// TIA Portal V17 export
// export: Created 2024-09-03T21:54:54.8850339Z, ExportSetting WithDefaults, DisplayName Totally Integrated Automation Portal, DisplayVersion V17 Update 7, DisplayName TIA Portal Openness, DisplayVersion V17 Update 7, DisplayName TIA Portal Version Control Interface, DisplayVersion V17, DisplayName SINAMICS Startdrive Advanced, DisplayVersion V17 SP2, DisplayName SINAMICS Startdrive G110M, G120, G120C, G120D, G120P, G115D, DisplayVersion V17 SP2, DisplayName SINAMICS Startdrive G130, G150, S120, S150, SINAMICS MV, S210, DisplayVersion V17 SP2, DisplayName STEP 7 Professional, DisplayVersion V17 Update 7, DisplayName STEP 7 Safety, DisplayVersion V17 Update 6, DisplayName WinCC Advanced / Unified PC, DisplayVersion V17 Update 7
DATA_BLOCK "DB_ProductionProgramList"   // DB6100
{ S7_Optimized_Access := 'FALSE' }
VERSION : 0.1
// stored: AutoNumber false, DBAccessibleFromOPCUA true, DBAccessibleFromWebserver true, IsOnlyStoredInLoadMemory false, IsWriteProtectedInAS false
   VAR RETAIN
      Program { S7_SetPoint := 'True'} : Array[1.."NumberOfProductionPrograms"] of "UDT_ProductionProgram";
   END_VAR
BEGIN
   Program[1]."Name" := 'LH-6 way';
   Program[2]."Name" := 'RH-6 way';
   Program[3]."Name" := 'LH-4 way';
   Program[4]."Name" := 'RH-4 way';
   Program[5]."Name" := 'startup';
   Program[6]."Name" := 'startup RH';
   Program[7..8]."Name" := '';
   Program[1].CupformingParametersLeft.DigiforceProgram := 1;
   Program[2].CupformingParametersLeft.DigiforceProgram := 2;
   Program[3].CupformingParametersLeft.DigiforceProgram := 1;
   Program[4].CupformingParametersLeft.DigiforceProgram := 2;
   Program[5..6].CupformingParametersLeft.DigiforceProgram := 1;
   Program[7..8].CupformingParametersLeft.DigiforceProgram := 0;
   Program[1..2].CupformingParametersLeft.FinalSpeed := 30.0;
   Program[3].CupformingParametersLeft.FinalSpeed := 20.0;
   Program[4].CupformingParametersLeft.FinalSpeed := 30.0;
   Program[5].CupformingParametersLeft.FinalSpeed := 25.0;
   Program[6].CupformingParametersLeft.FinalSpeed := 20.0;
   Program[7..8].CupformingParametersLeft.FinalSpeed := 0.0;
   Program[1..2].CupformingParametersLeft.ApproachSpeed := 95.0;
   Program[3].CupformingParametersLeft.ApproachSpeed := 100.0;
   Program[4].CupformingParametersLeft.ApproachSpeed := 95.0;
   Program[5].CupformingParametersLeft.ApproachSpeed := 25.0;
   Program[6].CupformingParametersLeft.ApproachSpeed := 100.0;
   Program[7..8].CupformingParametersLeft.ApproachSpeed := 0.0;
   Program[1..4].CupformingParametersLeft.FinalForce := 90.0;
   Program[5].CupformingParametersLeft.FinalForce := 10.0;
   Program[6].CupformingParametersLeft.FinalForce := 90.0;
   Program[7..8].CupformingParametersLeft.FinalForce := 0.0;
   Program[1..4].CupformingParametersLeft.ApproachForce := 20.0;
   Program[5].CupformingParametersLeft.ApproachForce := 10.0;
   Program[6].CupformingParametersLeft.ApproachForce := 20.0;
   Program[7..8].CupformingParametersLeft.ApproachForce := 0.0;
   Program[1..4].CupformingParametersLeft.EndWayImmediate := 7.5;
   Program[5].CupformingParametersLeft.EndWayImmediate := 2.55;
   Program[6].CupformingParametersLeft.EndWayImmediate := 9.9;
   Program[7..8].CupformingParametersLeft.EndWayImmediate := 0.0;
   Program[1..4].CupformingParametersLeft.EndWayWithTimeout := 8.6;
   Program[5].CupformingParametersLeft.EndWayWithTimeout := 3.0;
   Program[6].CupformingParametersLeft.EndWayWithTimeout := 9.9;
   Program[7..8].CupformingParametersLeft.EndWayWithTimeout := 0.0;
   Program[1..4].CupformingParametersLeft.SwitchingWay := 50.0;
   Program[5].CupformingParametersLeft.SwitchingWay := 20.0;
   Program[6].CupformingParametersLeft.SwitchingWay := 50.0;
   Program[7..8].CupformingParametersLeft.SwitchingWay := 0.0;
   Program[1..5].CupformingParametersLeft.EndWayTimeout := T#300MS;
   Program[6].CupformingParametersLeft.EndWayTimeout := T#200MS;
   Program[7..8].CupformingParametersLeft.EndWayTimeout := T#0MS;
   Program[1].CupformingParametersRight.DigiforceProgram := 1;
   Program[2].CupformingParametersRight.DigiforceProgram := 2;
   Program[3].CupformingParametersRight.DigiforceProgram := 1;
   Program[4].CupformingParametersRight.DigiforceProgram := 2;
   Program[5..6].CupformingParametersRight.DigiforceProgram := 1;
   Program[7..8].CupformingParametersRight.DigiforceProgram := 0;
   Program[1..4].CupformingParametersRight.FinalSpeed := 30.0;
   Program[5].CupformingParametersRight.FinalSpeed := 25.0;
   Program[6].CupformingParametersRight.FinalSpeed := 20.0;
   Program[7..8].CupformingParametersRight.FinalSpeed := 0.0;
   Program[1..2].CupformingParametersRight.ApproachSpeed := 100.0;
   Program[3].CupformingParametersRight.ApproachSpeed := 95.0;
   Program[4].CupformingParametersRight.ApproachSpeed := 100.0;
   Program[5].CupformingParametersRight.ApproachSpeed := 25.0;
   Program[6].CupformingParametersRight.ApproachSpeed := 100.0;
   Program[7..8].CupformingParametersRight.ApproachSpeed := 0.0;
   Program[1..6].CupformingParametersRight.FinalForce := 60.0;
   Program[7..8].CupformingParametersRight.FinalForce := 0.0;
   Program[1..6].CupformingParametersRight.ApproachForce := 10.0;
   Program[7..8].CupformingParametersRight.ApproachForce := 0.0;
   Program[1..4].CupformingParametersRight.EndWayImmediate := 7.8;
   Program[5].CupformingParametersRight.EndWayImmediate := 2.7;
   Program[6].CupformingParametersRight.EndWayImmediate := 9.9;
   Program[7..8].CupformingParametersRight.EndWayImmediate := 0.0;
   Program[1..2].CupformingParametersRight.EndWayWithTimeout := 8.4;
   Program[3].CupformingParametersRight.EndWayWithTimeout := 8.6;
   Program[4].CupformingParametersRight.EndWayWithTimeout := 8.4;
   Program[5].CupformingParametersRight.EndWayWithTimeout := 3.0;
   Program[6].CupformingParametersRight.EndWayWithTimeout := 9.9;
   Program[7..8].CupformingParametersRight.EndWayWithTimeout := 0.0;
   Program[1..4].CupformingParametersRight.SwitchingWay := 50.0;
   Program[5].CupformingParametersRight.SwitchingWay := 20.0;
   Program[6].CupformingParametersRight.SwitchingWay := 50.0;
   Program[7..8].CupformingParametersRight.SwitchingWay := 0.0;
   Program[1..4].CupformingParametersRight.EndWayTimeout := T#1S;
   Program[5].CupformingParametersRight.EndWayTimeout := T#300MS;
   Program[6].CupformingParametersRight.EndWayTimeout := T#200MS;
   Program[7..8].CupformingParametersRight.EndWayTimeout := T#0MS;
   Program[1].St1Insertion[1..6] := TRUE;
   Program[1].St1Insertion[7..20] := FALSE;
   Program[2].St1Insertion[1..6] := TRUE;
   Program[2].St1Insertion[7..20] := FALSE;
   Program[3].St1Insertion[1..2] := TRUE;
   Program[3].St1Insertion[3] := FALSE;
   Program[3].St1Insertion[4..6] := TRUE;
   Program[3].St1Insertion[7..20] := FALSE;
   Program[4].St1Insertion[1..5] := TRUE;
   Program[4].St1Insertion[6..20] := FALSE;
   Program[5].St1Insertion[1] := TRUE;
   Program[5].St1Insertion[2] := FALSE;
   Program[5].St1Insertion[3..5] := TRUE;
   Program[5].St1Insertion[6] := FALSE;
   Program[5].St1Insertion[7] := TRUE;
   Program[5].St1Insertion[8] := FALSE;
   Program[5].St1Insertion[9..10] := TRUE;
   Program[5].St1Insertion[11] := FALSE;
   Program[5].St1Insertion[12..17] := TRUE;
   Program[5].St1Insertion[18] := FALSE;
   Program[5].St1Insertion[19] := TRUE;
   Program[5].St1Insertion[20] := FALSE;
   Program[6].St1Insertion[1..4] := TRUE;
   Program[6].St1Insertion[5..20] := FALSE;
   Program[7].St1Insertion[1..20] := FALSE;
   Program[8].St1Insertion[1..20] := FALSE;
   Program[1].St1InsertionUsed[1..6] := TRUE;
   Program[1].St1InsertionUsed[7..20] := FALSE;
   Program[2].St1InsertionUsed[1..6] := TRUE;
   Program[2].St1InsertionUsed[7..20] := FALSE;
   Program[3].St1InsertionUsed[1..2] := TRUE;
   Program[3].St1InsertionUsed[3] := FALSE;
   Program[3].St1InsertionUsed[4..6] := TRUE;
   Program[3].St1InsertionUsed[7..20] := FALSE;
   Program[4].St1InsertionUsed[1..5] := TRUE;
   Program[4].St1InsertionUsed[6..20] := FALSE;
   Program[5].St1InsertionUsed[1..7] := TRUE;
   Program[5].St1InsertionUsed[8] := FALSE;
   Program[5].St1InsertionUsed[9..19] := TRUE;
   Program[5].St1InsertionUsed[20] := FALSE;
   Program[6].St1InsertionUsed[1..4] := TRUE;
   Program[6].St1InsertionUsed[5..20] := FALSE;
   Program[7].St1InsertionUsed[1..20] := FALSE;
   Program[8].St1InsertionUsed[1..20] := FALSE;
   Program[1].FaureciaNumber := '2824317X';
   Program[2].FaureciaNumber := '2841135X';
   Program[3].FaureciaNumber := '2824317X';
   Program[4].FaureciaNumber := '2841135X';
   Program[5].FaureciaNumber := '2567208X';
   Program[6].FaureciaNumber := 'xxxx';
   Program[7..8].FaureciaNumber := '';
   Program[1..6].FaureciaNumberStartChar := 9;
   Program[7..8].FaureciaNumberStartChar := 0;
   Program[1..6].FaureciaNumberLength := 8;
   Program[7..8].FaureciaNumberLength := 0;
   Program[1].MechanicalType := 0;
   Program[2].MechanicalType := 1;
   Program[3].MechanicalType := 0;
   Program[4].MechanicalType := 1;
   Program[5].MechanicalType := 0;
   Program[6].MechanicalType := 1;
   Program[7..8].MechanicalType := 0;
   Program[1].Camera_program[0] := 0;
   Program[1].Camera_program[1..4] := 1;
   Program[2].Camera_program[0..4] := 0;
   Program[3].Camera_program[0] := 0;
   Program[3].Camera_program[1] := 1;
   Program[3].Camera_program[2..3] := 3;
   Program[3].Camera_program[4] := 1;
   Program[4].Camera_program[0..4] := 0;
   Program[5].Camera_program[0..4] := 0;
   Program[6].Camera_program[0..4] := 0;
   Program[7].Camera_program[0..1] := 0;
   Program[7].Camera_program[2..3] := 4;
   Program[7].Camera_program[4] := 0;
   Program[8].Camera_program[0..4] := 0;
   Program[1].Riveting_program_left[0] := 0;
   Program[1].Riveting_program_left[1..2] := 1;
   Program[2].Riveting_program_left[0] := 0;
   Program[2].Riveting_program_left[1] := 3;
   Program[2].Riveting_program_left[2] := 1;
   Program[3].Riveting_program_left[0] := 0;
   Program[3].Riveting_program_left[1] := 3;
   Program[3].Riveting_program_left[2] := 1;
   Program[4].Riveting_program_left[0] := 0;
   Program[4].Riveting_program_left[1] := 3;
   Program[4].Riveting_program_left[2] := 1;
   Program[5].Riveting_program_left[0..2] := 0;
   Program[6].Riveting_program_left[0] := 0;
   Program[6].Riveting_program_left[1..2] := 2;
   Program[7].Riveting_program_left[0..2] := 0;
   Program[8].Riveting_program_left[0..2] := 0;
   Program[1].Riveting_program_right[0] := 0;
   Program[1].Riveting_program_right[1..2] := 1;
   Program[2].Riveting_program_right[0] := 0;
   Program[2].Riveting_program_right[1..2] := 1;
   Program[3].Riveting_program_right[0] := 0;
   Program[3].Riveting_program_right[1] := 3;
   Program[3].Riveting_program_right[2] := 1;
   Program[4].Riveting_program_right[0] := 0;
   Program[4].Riveting_program_right[1] := 3;
   Program[4].Riveting_program_right[2] := 1;
   Program[5].Riveting_program_right[0..2] := 0;
   Program[6].Riveting_program_right[0] := 0;
   Program[6].Riveting_program_right[1..2] := 2;
   Program[7].Riveting_program_right[0..2] := 0;
   Program[8].Riveting_program_right[0..2] := 0;
   Program[1..2].Total_number_of_rivets_4 := TRUE;
   Program[3..5].Total_number_of_rivets_4 := FALSE;
   Program[6].Total_number_of_rivets_4 := TRUE;
   Program[7..8].Total_number_of_rivets_4 := FALSE;
   Program[1..8].NumberOfReadings := 0;
   Program[1].Readings[1..4].Enable := FALSE;
   Program[2].Readings[1..4].Enable := FALSE;
   Program[3].Readings[1..4].Enable := FALSE;
   Program[4].Readings[1..4].Enable := FALSE;
   Program[5].Readings[1..4].Enable := FALSE;
   Program[6].Readings[1..4].Enable := FALSE;
   Program[7].Readings[1..4].Enable := FALSE;
   Program[8].Readings[1..4].Enable := FALSE;
   Program[1].Readings[1..4].ReaderNumber := 0;
   Program[2].Readings[1..4].ReaderNumber := 0;
   Program[3].Readings[1..4].ReaderNumber := 0;
   Program[4].Readings[1..4].ReaderNumber := 0;
   Program[5].Readings[1..4].ReaderNumber := 0;
   Program[6].Readings[1..4].ReaderNumber := 0;
   Program[7].Readings[1..4].ReaderNumber := 0;
   Program[8].Readings[1..4].ReaderNumber := 0;
   Program[1].Readings[1..4]."Name" := WSTRING#'';
   Program[2].Readings[1..4]."Name" := WSTRING#'';
   Program[3].Readings[1..4]."Name" := WSTRING#'';
   Program[4].Readings[1..4]."Name" := WSTRING#'';
   Program[5].Readings[1..4]."Name" := WSTRING#'';
   Program[6].Readings[1..4]."Name" := WSTRING#'';
   Program[7].Readings[1..4]."Name" := WSTRING#'';
   Program[8].Readings[1..4]."Name" := WSTRING#'';
   Program[1].Readings[1..4].LabelType := 0;
   Program[2].Readings[1..4].LabelType := 0;
   Program[3].Readings[1..4].LabelType := 0;
   Program[4].Readings[1..4].LabelType := 0;
   Program[5].Readings[1..4].LabelType := 0;
   Program[6].Readings[1..4].LabelType := 0;
   Program[7].Readings[1..4].LabelType := 0;
   Program[8].Readings[1..4].LabelType := 0;
   Program[1].Readings[1..4].ReferenceToFound := WSTRING#'';
   Program[2].Readings[1..4].ReferenceToFound := WSTRING#'';
   Program[3].Readings[1..4].ReferenceToFound := WSTRING#'';
   Program[4].Readings[1..4].ReferenceToFound := WSTRING#'';
   Program[5].Readings[1..4].ReferenceToFound := WSTRING#'';
   Program[6].Readings[1..4].ReferenceToFound := WSTRING#'';
   Program[7].Readings[1..4].ReferenceToFound := WSTRING#'';
   Program[8].Readings[1..4].ReferenceToFound := WSTRING#'';
   Program[1].Readings[1..4].ReferenceStartPosition := 0;
   Program[2].Readings[1..4].ReferenceStartPosition := 0;
   Program[3].Readings[1..4].ReferenceStartPosition := 0;
   Program[4].Readings[1..4].ReferenceStartPosition := 0;
   Program[5].Readings[1..4].ReferenceStartPosition := 0;
   Program[6].Readings[1..4].ReferenceStartPosition := 0;
   Program[7].Readings[1..4].ReferenceStartPosition := 0;
   Program[8].Readings[1..4].ReferenceStartPosition := 0;
   Program[1].Readings[1..4].ReferenceLenght := 0;
   Program[2].Readings[1..4].ReferenceLenght := 0;
   Program[3].Readings[1..4].ReferenceLenght := 0;
   Program[4].Readings[1..4].ReferenceLenght := 0;
   Program[5].Readings[1..4].ReferenceLenght := 0;
   Program[6].Readings[1..4].ReferenceLenght := 0;
   Program[7].Readings[1..4].ReferenceLenght := 0;
   Program[8].Readings[1..4].ReferenceLenght := 0;
   Program[1].Readings[1..4].MasterReadingNumber := 0;
   Program[2].Readings[1..4].MasterReadingNumber := 0;
   Program[3].Readings[1..4].MasterReadingNumber := 0;
   Program[4].Readings[1..4].MasterReadingNumber := 0;
   Program[5].Readings[1..4].MasterReadingNumber := 0;
   Program[6].Readings[1..4].MasterReadingNumber := 0;
   Program[7].Readings[1..4].MasterReadingNumber := 0;
   Program[8].Readings[1..4].MasterReadingNumber := 0;
   Program[1].Readings[1..4].LinkedMasterNumber := 0;
   Program[2].Readings[1..4].LinkedMasterNumber := 0;
   Program[3].Readings[1..4].LinkedMasterNumber := 0;
   Program[4].Readings[1..4].LinkedMasterNumber := 0;
   Program[5].Readings[1..4].LinkedMasterNumber := 0;
   Program[6].Readings[1..4].LinkedMasterNumber := 0;
   Program[7].Readings[1..4].LinkedMasterNumber := 0;
   Program[8].Readings[1..4].LinkedMasterNumber := 0;
   Program[1].Readings[1].Message[1..6].MessageType := 0;
   Program[1].Readings[2].Message[1..6].MessageType := 0;
   Program[1].Readings[3].Message[1..6].MessageType := 0;
   Program[1].Readings[4].Message[1..6].MessageType := 0;
   Program[2].Readings[1].Message[1..6].MessageType := 0;
   Program[2].Readings[2].Message[1..6].MessageType := 0;
   Program[2].Readings[3].Message[1..6].MessageType := 0;
   Program[2].Readings[4].Message[1..6].MessageType := 0;
   Program[3].Readings[1].Message[1..6].MessageType := 0;
   Program[3].Readings[2].Message[1..6].MessageType := 0;
   Program[3].Readings[3].Message[1..6].MessageType := 0;
   Program[3].Readings[4].Message[1..6].MessageType := 0;
   Program[4].Readings[1].Message[1..6].MessageType := 0;
   Program[4].Readings[2].Message[1..6].MessageType := 0;
   Program[4].Readings[3].Message[1..6].MessageType := 0;
   Program[4].Readings[4].Message[1..6].MessageType := 0;
   Program[5].Readings[1].Message[1..6].MessageType := 0;
   Program[5].Readings[2].Message[1..6].MessageType := 0;
   Program[5].Readings[3].Message[1..6].MessageType := 0;
   Program[5].Readings[4].Message[1..6].MessageType := 0;
   Program[6].Readings[1].Message[1..6].MessageType := 0;
   Program[6].Readings[2].Message[1..6].MessageType := 0;
   Program[6].Readings[3].Message[1..6].MessageType := 0;
   Program[6].Readings[4].Message[1..6].MessageType := 0;
   Program[7].Readings[1].Message[1..6].MessageType := 0;
   Program[7].Readings[2].Message[1..6].MessageType := 0;
   Program[7].Readings[3].Message[1..6].MessageType := 0;
   Program[7].Readings[4].Message[1..6].MessageType := 0;
   Program[8].Readings[1].Message[1..6].MessageType := 0;
   Program[8].Readings[2].Message[1..6].MessageType := 0;
   Program[8].Readings[3].Message[1..6].MessageType := 0;
   Program[8].Readings[4].Message[1..6].MessageType := 0;
   Program[1].Readings[1].Message[1..6].MessageFlagNumber := 0;
   Program[1].Readings[2].Message[1..6].MessageFlagNumber := 0;
   Program[1].Readings[3].Message[1..6].MessageFlagNumber := 0;
   Program[1].Readings[4].Message[1..6].MessageFlagNumber := 0;
   Program[2].Readings[1].Message[1..6].MessageFlagNumber := 0;
   Program[2].Readings[2].Message[1..6].MessageFlagNumber := 0;
   Program[2].Readings[3].Message[1..6].MessageFlagNumber := 0;
   Program[2].Readings[4].Message[1..6].MessageFlagNumber := 0;
   Program[3].Readings[1].Message[1..6].MessageFlagNumber := 0;
   Program[3].Readings[2].Message[1..6].MessageFlagNumber := 0;
   Program[3].Readings[3].Message[1..6].MessageFlagNumber := 0;
   Program[3].Readings[4].Message[1..6].MessageFlagNumber := 0;
   Program[4].Readings[1].Message[1..6].MessageFlagNumber := 0;
   Program[4].Readings[2].Message[1..6].MessageFlagNumber := 0;
   Program[4].Readings[3].Message[1..6].MessageFlagNumber := 0;
   Program[4].Readings[4].Message[1..6].MessageFlagNumber := 0;
   Program[5].Readings[1].Message[1..6].MessageFlagNumber := 0;
   Program[5].Readings[2].Message[1..6].MessageFlagNumber := 0;
   Program[5].Readings[3].Message[1..6].MessageFlagNumber := 0;
   Program[5].Readings[4].Message[1..6].MessageFlagNumber := 0;
   Program[6].Readings[1].Message[1..6].MessageFlagNumber := 0;
   Program[6].Readings[2].Message[1..6].MessageFlagNumber := 0;
   Program[6].Readings[3].Message[1..6].MessageFlagNumber := 0;
   Program[6].Readings[4].Message[1..6].MessageFlagNumber := 0;
   Program[7].Readings[1].Message[1..6].MessageFlagNumber := 0;
   Program[7].Readings[2].Message[1..6].MessageFlagNumber := 0;
   Program[7].Readings[3].Message[1..6].MessageFlagNumber := 0;
   Program[7].Readings[4].Message[1..6].MessageFlagNumber := 0;
   Program[8].Readings[1].Message[1..6].MessageFlagNumber := 0;
   Program[8].Readings[2].Message[1..6].MessageFlagNumber := 0;
   Program[8].Readings[3].Message[1..6].MessageFlagNumber := 0;
   Program[8].Readings[4].Message[1..6].MessageFlagNumber := 0;
END_DATA_BLOCK
